// TIA Portal V16 export
// export: Created 2023-03-29T11:03:26.3607854Z, ExportSetting WithDefaults, DisplayName Totally Integrated Automation Portal, DisplayVersion V16 Update 6, DisplayName TIA Portal Version Control Interface, DisplayVersion V16 Update 2, DisplayName TIA Portal Openness, DisplayVersion V16 Update 6, DisplayName STEP 7 Professional, DisplayVersion V16 Update 6, DisplayName STEP 7 Safety, DisplayVersion V16, DisplayName WinCC Advanced, DisplayVersion V16 Update 6
DATA_BLOCK "dbHold_download"   // DB58
TITLE = Instancja danych serwera TCP
{ S7_Optimized_Access := 'FALSE' }
AUTHOR : rtecmer
VERSION : 0.1
// Instancja dla funkcji Modbus TCP. Blok danych przechowujący dane pobrane z PLC Pompownia (zadane )
// stored: AutoNumber false, DBAccessibleFromOPCUA true, IsOnlyStoredInLoadMemory false, IsWriteProtectedInAS false
   VAR
      sterowanie : Struct
         act_położenie_Z10 : Word;   // Położenie zasuwy Z10 [%]
         set_poziom_napełniania : Real;   // wartość zadana poziomu napełniania
         set_poziom_opróżniania : Real;   // wartość zadana poziomu opróżniania
         set_res_bity_sterowania_napęami_1 : Word;   // bity sterowania napędami
         set_res_bity_sterowania_napęami_2 : Word := 16#0;   // bity sterowania napędami
         set_res_bity_tryb_napędów_1 : Word;   // bity sterowania przełączaniem trybów pracy
         set_res_bity_tryb_napędów_2 : Word := 16#0;   // bity sterowania przełączaniem trybów pracy
         rez_alarm_napędów : Word;   // bity kasowania alarmów napędów
         set_strategia_sterowania : Word;   // 0 - wyłączone, 1- Dosilanie, 2- Przetłaczanie, 3 - Automat
         set_sterowanie_cyklem : Word;   // 0- wyłączone, 1-Dobowe, 2- Tygodniowe, 3- Ręczne
         set_położenie_Z10 : Word;   // Położenie zasuwy Z10 [%]
         komunikacjaPLC : Word;   // kontrola komunikacji wysyłanie -PLC2 - PLC1
         set_magistrala_alarm_min_bar : Real;   // ciśnienie alarmu awaria na magistrali B5
      END_STRUCT;
      SendingTimes : Struct
         start_napełnianie : DTL;
         Stop_napełnianie : DTL;
         Start_przetłaczanie_1 : DTL;
         Stop_przetłaczanie_1 : DTL;
         Start_dosilanie_1 : DTL;
         Stop_dosilanie_1 : DTL;
      END_STRUCT;
   END_VAR
BEGIN
END_DATA_BLOCK
